{attribute 'qualified_only'}
VAR_GLOBAL
	bResetIClk: BOOL;
	{attribute 'TcLinkTo' := 'TIIB[Rack#1A-02 SFIN (EL1918)]^StandardInputs^Standard Out Var 18'}
	bESTOP AT %I*: BOOL;
	
	{attribute 'TcLinkTo' := 'TIIB[Rack#2B-05 SV_AIR (EL2004)]^Channel 1^Output'}
	bOpenSV1 AT %Q*: BOOL;
	{attribute 'TcLinkTo' := 'TIIB[Rack#2B-05 SV_AIR (EL2004)]^Channel 2^Output'}
	bOpenSV2 AT %Q*: BOOL;
	
	{attribute 'TcLinkTo' := 'TIIB[Rack#1C_ServoDR (NCR-HD Series)]^260th receive PDO Mapping^Positive torque limit value'}
	iServoTorqueLimitPositive AT %Q*: UINT;
	
	{attribute 'TcLinkTo' := 'TIIB[Rack#1C_ServoDR (NCR-HD Series)]^260th receive PDO Mapping^Negative torque limit value'}
	iServoTorqueLimitNegative AT %Q*: UINT;

	// 2Theta Servo
	// TIID^CX2020 (EtherCAT)^Term 1 (EK1200)^Term 2 (EK1122)^Rack#1C_ServoDR (NCR-HD Series)^260th transmit PDO Mapping^Digital inputs
	{attribute 'TcLinkTo' := 'TIIB[Rack#1C_ServoDR (NCR-HD Series)]^260th transmit PDO Mapping^Digital inputs'}
	i_ServoLimits AT %I* :UDINT;

	//TIIB[Rack#1C_ServoDR (NCR-HD Series)]^260th transmit PDO Mapping^Position actual value
	
	{attribute 'TcLinkTo' := '	.nRawEncoderULINT     	:= TIIB[Rack#1C_ServoDR (NCR-HD Series)]^260th transmit PDO Mapping^Position actual value
                                .bBrakeRelease			:= TIIB[Rack#1A-05 MB_2Th (EL2602)]^Channel 1^Output
	'}
	M1: DUT_MotionStage;
	
	// 2Theta Stepper
	//{attribute 'TcLinkTo' := '  .bBrakeRelease			:= TIIB[Rack#1A-05 MB_2Th (EL2602)]^Channel 1^Output'}
	M2: DUT_MotionStage;
	
	// XS1
	{attribute 'TcLinkTo' := '	.bLimitForwardEnable  	:= TIIB[Rack#2A-03 DR_XS1 (EL7041-0052)]^STM Status^Status^Digital input 1;
								.bLimitBackwardEnable 	:= TIIB[Rack#2A-03 DR_XS1 (EL7041-0052)]^STM Status^Status^Digital input 2;
								.nRawEncoderULINT     	:= TIIB[Rack#2B-07 ENC_X1_X2 (EL5042)]^FB Inputs Channel 1^Position
	'}
    M3: DUT_MotionStage;
	
	// XS2
	{attribute 'TcLinkTo' := '	.bLimitForwardEnable  	:= TIIB[Rack#2A-04 DR_XS2 (EL7041-0052)]^STM Status^Status^Digital input 1;
								.bLimitBackwardEnable 	:= TIIB[Rack#2A-04 DR_XS2 (EL7041-0052)]^STM Status^Status^Digital input 2;
								.nRawEncoderULINT     	:= TIIB[Rack#2B-07 ENC_X1_X2 (EL5042)]^FB Inputs Channel 2^Position
	'}
    M4: DUT_MotionStage;
	
	// YS1
	{attribute 'TcLinkTo' := '	.bLimitForwardEnable  	:= TIIB[Rack#2A-05 DR_YS1 (EL7041-0052)]^STM Status^Status^Digital input 1;
								.bLimitBackwardEnable 	:= TIIB[Rack#2A-05 DR_YS1 (EL7041-0052)]^STM Status^Status^Digital input 2;
								.nRawEncoderULINT     	:= TIIB[Rack#2B-08 ENC_Y1_Y2 (EL5042)]^FB Inputs Channel 1^Position
	'}
    M5: DUT_MotionStage;
	
	// YS2
	{attribute 'TcLinkTo' := '	.bLimitForwardEnable  	:= TIIB[Rack#2A-06 DR_YS2 (EL7041-0052)]^STM Status^Status^Digital input 1;
								.bLimitBackwardEnable 	:= TIIB[Rack#2A-06 DR_YS2 (EL7041-0052)]^STM Status^Status^Digital input 2;
								.nRawEncoderULINT     	:= TIIB[Rack#2B-08 ENC_Y1_Y2 (EL5042)]^FB Inputs Channel 1^Position
	'}
    M6: DUT_MotionStage;
	
	// YG1
    {attribute 'TcLinkTo' := '	.bLimitForwardEnable	:= TIIB[Rack#2A-10 DR_YG1 (EL7041-0052)]^STM Status^Status^Digital input 1;
								.bLimitBackwardEnable	:= TIIB[Rack#2A-10 DR_YG1 (EL7041-0052)]^STM Status^Status^Digital input 2;
								.nRawEncoderULINT		:= TIIB[Rack#2B-10 ENC_YG1_YG2 (EL5042)]^FB Inputs Channel 1^Position
	'}
	M7: DUT_MotionStage;
	
	// YG2
    {attribute 'TcLinkTo' := '	.bLimitForwardEnable	:= TIIB[Rack#2A-11 DR_YG2 (EL7041-0052)]^STM Status^Status^Digital input 1;
								.bLimitBackwardEnable	:= TIIB[Rack#2A-11 DR_YG2 (EL7041-0052)]^STM Status^Status^Digital input 2;
								.nRawEncoderULINT		:= TIIB[Rack#2B-10 ENC_YG1_YG2 (EL5042)]^FB Inputs Channel 2^Position
	'}
    M8: DUT_MotionStage;
	
	// YG3
    {attribute 'TcLinkTo' := '	.bLimitForwardEnable	:= TIIB[Rack#2A-12 DR_YG3 (EL7041-0052)]^STM Status^Status^Digital input 1;
								.bLimitBackwardEnable	:= TIIB[Rack#2A-12 DR_YG3 (EL7041-0052)]^STM Status^Status^Digital input 2;
								.nRawEncoderULINT		:= TIIB[Rack#2B-11 ENC_YG3_X1PM (EL5042)]^FB Inputs Channel 1^Position
	'}
    M9: DUT_MotionStage;
	
	
	// RxG
    {attribute 'TcLinkTo' := '	.bLimitForwardEnable	:= TIIB[Rack#2A-08 DR_RxG (EL7041-0052)]^STM Status^Status^Digital input 1;
								.bLimitBackwardEnable	:= TIIB[Rack#2A-08 DR_RxG (EL7041-0052)]^STM Status^Status^Digital input 2;
								.nRawEncoderULINT		:= TIIB[Rack#2B-09 ENC_RxG_XG (EL5042)]^FB Inputs Channel 1 compact^Position
	'}
    M10: DUT_MotionStage;
	
	// XG
    {attribute 'TcLinkTo' := '	.bLimitForwardEnable	:= TIIB[Rack#2A-09 DR_XG (EL7041-0052)]^STM Status^Status^Digital input 1;
								.bLimitBackwardEnable	:= TIIB[Rack#2A-09 DR_XG (EL7041-0052)]^STM Status^Status^Digital input 2;
								.nRawEncoderULINT		:= TIIB[Rack#2B-09 ENC_RxG_XG (EL5042)]^FB Inputs Channel 2^Position
	'}
    M11: DUT_MotionStage;
	
	// XPM1
    {attribute 'TcLinkTo' := '	.bLimitForwardEnable	:= TIIB[Rack#2A-14 DR_XPM1 (EL7041-0052)]^STM Status^Status^Digital input 1;
								.bLimitBackwardEnable	:= TIIB[Rack#2A-14 DR_XPM1 (EL7041-0052)]^STM Status^Status^Digital input 2;
								.nRawEncoderULINT		:= TIIB[Rack#2B-11 ENC_YG3_X1PM (EL5042)]^FB Inputs Channel 2^Position
	'}
    M12: DUT_MotionStage;
	
	// XPM2
    {attribute 'TcLinkTo' := '	.bLimitForwardEnable	:= TIIB[Rack#2A-15 DR_XPM2 (EL7041-0052)]^STM Status^Status^Digital input 1;
								.bLimitBackwardEnable	:= TIIB[Rack#2A-15 DR_XPM2 (EL7041-0052)]^STM Status^Status^Digital input 2;
								.nRawEncoderULINT		:= TIIB[Rack#2B-12 ENC_X2PM_RzPM (EL5042)]^FB Inputs Channel 1^Position
	'}
	M13: DUT_MotionStage;
	
	// RzPM
    {attribute 'TcLinkTo' := '	.bLimitForwardEnable	:= TIIB[Rack#2A-16 DR_RzPM (EL7041-0052)]^STM Status^Status^Digital input 1;
								.bLimitBackwardEnable	:= TIIB[Rack#2A-16 DR_RzPM (EL7041-0052)]^STM Status^Status^Digital input 2;
								.nRawEncoderULINT		:= TIIB[Rack#2B-12 ENC_X2PM_RzPM (EL5042)]^FB Inputs Channel 2^Position
	'}
    M14: DUT_MotionStage;

	// YDF1
	{attribute 'TcLinkTo' := '	.bLimitForwardEnable  	:= TIIB[Rack#2B-15 DR_YDF1 (EL7041-0052)]^STM Status^Status^Digital input 1;
								.bLimitBackwardEnable 	:= TIIB[Rack#2B-15 DR_YDF1 (EL7041-0052)]^STM Status^Status^Digital input 2
	'}
    M15: DUT_MotionStage;
	
	// YDF2
	{attribute 'TcLinkTo' := '	.bLimitForwardEnable  	:= TIIB[Rack#2B-16 DR_YDF2 (EL7041-0052)]^STM Status^Status^Digital input 1;
								.bLimitBackwardEnable 	:= TIIB[Rack#2B-16 DR_YDF2 (EL7041-0052)]^STM Status^Status^Digital input 2
	'}
    M16: DUT_MotionStage;
	
	// YDF3
	{attribute 'TcLinkTo' := '	.bLimitForwardEnable  	:= TIIB[Rack#2B-19 DR_YDF3 (EL7041-0052)]^STM Status^Status^Digital input 1;
								.bLimitBackwardEnable 	:= TIIB[Rack#2B-19 DR_YDF3 (EL7041-0052)]^STM Status^Status^Digital input 2
	'}
    M17: DUT_MotionStage;
	
	// XSDC1
	{attribute 'TcLinkTo' := '	.bLimitForwardEnable  	:= TIIB[BOX-09 DR_XSDC1 (EL7041-0052)]^STM Status^Status^Digital input 1;
								.bLimitBackwardEnable 	:= TIIB[BOX-09 DR_XSDC1 (EL7041-0052)]^STM Status^Status^Digital input 2;
								.nRawEncoderULINT     	:= TIIB[BOX-03 ENC_X1_X2 (EL5042)]^FB Inputs Channel 1^Position
	'}
    M18: DUT_MotionStage;
	
	// XSDC2
	{attribute 'TcLinkTo' := '	.bLimitForwardEnable	:= TIIB[BOX-10 DR_XSDC2 (EL7041-0052)]^STM Status^Status^Digital input 1;
								.bLimitBackwardEnable 	:= TIIB[BOX-10 DR_XSDC2 (EL7041-0052)]^STM Status^Status^Digital input 2;
								.nRawEncoderULINT     	:= TIIB[BOX-03 ENC_X1_X2 (EL5042)]^FB Inputs Channel 2^Position
	'}
    M19: DUT_MotionStage;
	
	// YSDC1
	{attribute 'TcLinkTo' := '	.bLimitForwardEnable	:= TIIB[BOX-11 DR_YSDC1 (EL7041-0052)]^STM Status^Status^Digital input 1;
								.bLimitBackwardEnable 	:= TIIB[BOX-11 DR_YSDC1 (EL7041-0052)]^STM Status^Status^Digital input 2;
								.nRawEncoderULINT     	:= TIIB[BOX-04 ENC_Y1_Y2 (EL5042)]^FB Inputs Channel 1^Position
	'}
    M20: DUT_MotionStage;
	
	// YSDC2
	{attribute 'TcLinkTo' := '	.bLimitForwardEnable	:= TIIB[BOX-12 DR_YSDC2 (EL7041-0052)]^STM Status^Status^Digital input 1;
								.bLimitBackwardEnable 	:= TIIB[BOX-12 DR_YSDC2 (EL7041-0052)]^STM Status^Status^Digital input 2;
								.nRawEncoderULINT     	:= TIIB[BOX-04 ENC_Y1_Y2 (EL5042)]^FB Inputs Channel 1^Position
	'}
    M21: DUT_MotionStage;

	// XDC
	{attribute 'TcLinkTo' := '	.bLimitForwardEnable  	:= TIIB[BOX-14 DR_XDC (EL7041-0052)]^STM Status^Status^Digital input 1;
								.bLimitBackwardEnable 	:= TIIB[BOX-14 DR_XDC (EL7041-0052)]^STM Status^Status^Digital input 2;
								.nRawEncoderULINT     	:= TIIB[BOX-05 ENC_XDC_RyDC (EL5042)]^FB Inputs Channel 1^Position
	'}
    M22: DUT_MotionStage;
	
	// RyDC
	{attribute 'TcLinkTo' := '	.bLimitForwardEnable	:= TIIB[BOX-15 DR_RyDC (EL7041-0052)]^STM Status^Status^Digital input 1;
								.bLimitBackwardEnable	:= TIIB[BOX-15 DR_RyDC (EL7041-0052)]^STM Status^Status^Digital input 2;
								.nRawEncoderULINT		:= TIIB[BOX-05 ENC_XDC_RyDC (EL5042)]^FB Inputs Channel 2^Position
	'}
    M23: DUT_MotionStage;
	
	// ZDC
	{attribute 'TcLinkTo' := '	.bLimitForwardEnable	:= TIIB[BOX-16 DR_ZDC (EL7041-0052)]^STM Status^Status^Digital input 1;
								.bLimitBackwardEnable	:= TIIB[BOX-16 DR_ZDC (EL7041-0052)]^STM Status^Status^Digital input 2;
								.nRawEncoderULINT		:= TIIB[BOX-06 ENC_ZDC_YF1 (EL5042)]^FB Inputs Channel 1^Position
	'}
    M24: DUT_MotionStage;

	// YF1
	{attribute 'TcLinkTo' := '	.bLimitForwardEnable	:= TIIB[Rack#1A-02 SFIN (EL1918)]^StandardInputs^Standard Out Var 10;
								.bLimitBackwardEnable 	:= TIIB[Rack#1A-02 SFIN (EL1918)]^StandardInputs^Standard Out Var 11;
								.nRawEncoderULINT     	:= TIIB[BOX-06 ENC_ZDC_YF1 (EL5042)]^FB Inputs Channel 2^Position;
								.bBrakeRelease        	:= TIIB[BOX-19 MB_YF1_YF2 (EL2602)]^Channel 1^Output
	'}
    M25: DUT_MotionStage;
	
	// YF2
	{attribute 'TcLinkTo' := '	.bLimitForwardEnable	:= TIIB[Rack#1A-02 SFIN (EL1918)]^StandardInputs^Standard Out Var 12;
								.bLimitBackwardEnable	:= TIIB[Rack#1A-02 SFIN (EL1918)]^StandardInputs^Standard Out Var 13;
								.nRawEncoderULINT     	:= TIIB[BOX-07 ENC_YF2_ZF (EL5042)]^FB Inputs Channel 1^Position;
								.bBrakeRelease			:= TIIB[BOX-19 MB_YF1_YF2 (EL2602)]^Channel 2^Output
	'}
	M26: DUT_MotionStage;
	
	// ZF
	{attribute 'TcLinkTo' := '	.bLimitForwardEnable	:= TIIB[Rack#1A-02 SFIN (EL1918)]^StandardInputs^Standard Out Var 14;
								.bLimitBackwardEnable	:= TIIB[Rack#1A-02 SFIN (EL1918)]^StandardInputs^Standard Out Var 15;
								.nRawEncoderULINT		:= TIIB[BOX-07 ENC_YF2_ZF (EL5042)]^FB Inputs Channel 2^Position;
								.bBrakeRelease			:= TIIB[Rack#2B-18 MB_ZF (EL2602)]^Channel 1^Output
	'}
	M27: DUT_MotionStage;
	
	
END_VAR

(* stored: Version 1.1.0.1, ProductVersion 3.1.4022.18
   GVL GVL_Main: Id {52c31e46-cb36-4543-bf43-ce4ccb700f52} *)
